// TIA Portal V16 export
// export: Created 2023-08-28T09:37:52.5008051Z, ExportSetting WithDefaults, DisplayName Totally Integrated Automation Portal, DisplayVersion V16 Update 6, DisplayName TIA Portal Version Control Interface, DisplayVersion V16 Update 2, DisplayName TIA Portal Openness, DisplayVersion V16 Update 6, DisplayName STEP 7 Professional, DisplayVersion V16 Update 6, DisplayName STEP 7 Safety, DisplayVersion V16, DisplayName WinCC Advanced, DisplayVersion V16 Update 6
DATA_BLOCK "KALMAN_DB"   // DB125
{ S7_Optimized_Access := 'TRUE' }
VERSION : 0.1
// stored: AutoNumber false, DBAccessibleFromOPCUA true, IsOnlyStoredInLoadMemory false, IsRetainMemResEnabled false, IsWriteProtectedInAS false, MemoryReserve 250
   VAR
      kalman_P : Array[0..4] of Real;
      kalman_K : Array[0..4] of Real;
      kalman_Q : Array[0..4] of Real;
      kalman_R : Array[0..4] of Real;
      kalman_napiecie : Array[0..4] of Real;
      pomiar_napiecie : Array[0..4] of Real;
      wejscie_anal : Array[0..4] of Word;
   END_VAR
BEGIN
   // kalman_napiecie[0] : ciśnienie B6 tłoczenie
   // kalman_napiecie[1] : ciśnienie B7 zasilania
   // kalman_napiecie[2] : ciśnienie B8 ssania
   // kalman_napiecie[3] : przepływ
   // pomiar_napiecie[0] : ciśnienie B6 tłoczenie
   // pomiar_napiecie[1] : ciśnienie B7 zasilania
   // pomiar_napiecie[2] : ciśnienie B8 ssania
   // pomiar_napiecie[3] : przepływ
END_DATA_BLOCK
